{attribute 'qualified_only'}
{attribute 'strict'}
{attribute 'to_string'}
TYPE eCommands :
(
	MoveL 			:=0,
	MoveJ			:=1,
	MoveLRelativ 	:=2,
	MoveJRelativ 	:=3,
	SetDO			:=4,
	ReadDI			:=5,
	MoveJJoints		:=6,
	NavigateToGoal	:=7,
	NavigateToPoint	:=8,
	Dock			:=9,
	Undock			:=10,
	Homing			:=11,
	StopMotion		:=12,
	
	
	//Generic predefined Controls, no settings needed
	MoveToHomePosition := 13,
	MoveToSafePosition := 14
	
	
	
);
END_TYPE

(* stored: Version 1.1.0.1, ProductVersion 3.1.4026.18
   DUT eCommands: Id {229201d8-2c42-4601-b776-bb44db293d9d} *)
